(* PLC project BlogProject.project, CODESYS CODESYS V3.5 SP14 Patch 3 *)
(* stored: creationDateTime 2021-10-07T21:03:34.5053147, modificationDateTime 2021-10-07T20:40:20.1109198 *)

VAR_GLOBAL  (* FactoryStateGVL *)
  StartCommand : BOOL;
  StopCommand : BOOL;
  SystemStartFeedBack : BOOL;
  SystemStopFeedBack : BOOL;
  isErrorReset : mcIsErrorReset;
  isSystemChecked : mcIsSystemChecked;
  isSystemError : mcIsSystemError;
  isSystemStartCommand : mcIsSystemStartCommand;
  isSystemStarted : mcIsSystemStarted;
  isSystemStopCommand : mcIsSystemStopCommand;
  isSystemStoped : mcIsSystemStoped;
  NoEvent : mcNoEvent;
  NoAction : mcNoAction;
  StartSystem : mcStartSystem;
  StopSystem : mcStopSystem;
  stateSystemOff : udtTransition := (eCurrentState := enumState.SYSTEM_OFF, mcEvent_1 := NoEvent, mcEvent_2 := isSystemStartCommand, mcAction_1 := NoAction, mcAction_2 := NoAction, eNextStage := enumState.SYSTEM_CHECK);
  stateSystemCheck1 : udtTransition := (eCurrentState := enumState.SYSTEM_CHECK, mcEvent_1 := NoEvent, mcEvent_2 := isSystemChecked, mcAction_1 := StartSystem, mcAction_2 := NoAction, eNextStage := enumState.SYSTEM_START);
  stateSystemCheck2 : udtTransition := (eCurrentState := enumState.SYSTEM_CHECK, mcEvent_1 := NoEvent, mcEvent_2 := isSystemError, mcAction_1 := NoAction, mcAction_2 := NoAction, eNextStage := enumState.SYSTEM_ERR);
  stateSystemStart1 : udtTransition := (eCurrentState := enumState.SYSTEM_START, mcEvent_1 := NoEvent, mcEvent_2 := isSystemStarted, mcAction_1 := NoAction, mcAction_2 := NoAction, eNextStage := enumState.SYSTEM_RUN);
  stateSystemStart2 : udtTransition := (eCurrentState := enumState.SYSTEM_START, mcEvent_1 := NoEvent, mcEvent_2 := isSystemError, mcAction_1 := StopSystem, mcAction_2 := NoAction, eNextStage := enumState.SYSTEM_ERR);
  stateSystemRun1 : udtTransition := (eCurrentState := enumState.SYSTEM_RUN, mcEvent_1 := NoEvent, mcEvent_2 := isSystemStopCommand, mcAction_1 := NoAction, mcAction_2 := StopSystem, eNextStage := enumState.SYSTEM_STOP);
  stateSystemRun2 : udtTransition := (eCurrentState := enumState.SYSTEM_RUN, mcEvent_1 := NoEvent, mcEvent_2 := isSystemError, mcAction_1 := NoAction, mcAction_2 := StopSystem, eNextStage := enumState.SYSTEM_ERR);
  stateSystemStop1 : udtTransition := (eCurrentState := enumState.SYSTEM_STOP, mcEvent_1 := NoEvent, mcEvent_2 := isSystemStoped, mcAction_1 := NoAction, mcAction_2 := NoAction, eNextStage := enumState.SYSTEM_OFF);
  stateSystemStop2 : udtTransition := (eCurrentState := enumState.SYSTEM_STOP, mcEvent_1 := NoEvent, mcEvent_2 := isSystemError, mcAction_1 := NoAction, mcAction_2 := NoAction, eNextStage := enumState.SYSTEM_ERR);
  stateSystemErr : udtTransition := (eCurrentState := enumState.SYSTEM_ERR, mcEvent_1 := NoEvent, mcEvent_2 := isErrorReset, mcAction_1 := NoAction, mcAction_2 := NoAction, eNextStage := enumState.SYSTEM_OFF);
  System1 : udtSystem := (eCurrentState := enumState.SYSTEM_OFF, arTransactions := [stateSystemOff, stateSystemCheck1, stateSystemCheck2, stateSystemStart1, stateSystemStart2, stateSystemRun1, stateSystemRun2, stateSystemStop1, stateSystemStop2, stateSystemErr]);
END_VAR
